// TIA Portal V21 export
TYPE "Std_UnitàDiMisura"
   STRUCT
      In : "Std_ValoreConUm";
      Hmi : Struct
         Converti : Bool;
         Calcola : Bool;
      END_STRUCT;
      Dati : Struct
         FattoreDiConversione : Real;
      END_STRUCT;
      Out : "Std_ValoreConUm";
   END_STRUCT;
END_TYPE
